(* PLC project HIBACIP, Skikda University HIBACIP CODESYS 3.5.16.50 *)
(* stored: creationDateTime 2026-06-10T00:00:00, modificationDateTime 2026-06-10T00:00:00 *)

FUNCTION_BLOCK FB_SensorDiag
  VAR_INPUT
    w_RawAI : WORD;
    r_EU_Lo : REAL;
    r_EU_Hi : REAL;
    r_Filter_Alpha : REAL := 0.15;
    r_WB_Threshold : REAL := 1000.0;
  END_VAR
  VAR_OUTPUT
    r_ScaledPV : REAL;
    r_FilteredPV : REAL;
    b_WireFault : BOOL;
    b_BadQuality : BOOL;
  END_VAR
  VAR
    r_Raw : REAL;
    r_PrevFilt : REAL;
  END_VAR

            r_Raw := WORD_TO_REAL(w_RawAI);
IF r_Raw < r_WB_Threshold THEN
    b_WireFault  := TRUE;
    b_BadQuality := TRUE;
    r_ScaledPV   := -999.0;
    r_FilteredPV := -999.0;
    RETURN;
END_IF
b_WireFault := FALSE;
r_ScaledPV  := (r_Raw / 32767.0) * (r_EU_Hi - r_EU_Lo) + r_EU_Lo;
IF r_ScaledPV > r_EU_Hi THEN r_ScaledPV := r_EU_Hi; END_IF
IF r_ScaledPV < r_EU_Lo THEN r_ScaledPV := r_EU_Lo; END_IF
r_FilteredPV := r_Filter_Alpha * r_ScaledPV
    + (1.0 - r_Filter_Alpha) * r_PrevFilt;
r_PrevFilt   := r_FilteredPV;
b_BadQuality := b_WireFault;
          
END_FUNCTION_BLOCK

FUNCTION_BLOCK FB_ValveControl
  VAR_INPUT
    b_Open_Cmd : BOOL;
    b_EStop : BOOL;
    b_FailOpen : BOOL := FALSE;
  END_VAR
  VAR_OUTPUT
    q_ValveCoil : BOOL;
  END_VAR

            IF b_EStop THEN
    q_ValveCoil := b_FailOpen;
    RETURN;
END_IF
q_ValveCoil := b_Open_Cmd;
          
END_FUNCTION_BLOCK

FUNCTION_BLOCK FB_PumpControl
  VAR_INPUT
    b_Start_Cmd : BOOL;
    b_Overload_OK : BOOL;
    b_EStop : BOOL;
  END_VAR
  VAR_OUTPUT
    q_PumpCoil : BOOL;
    b_Running : BOOL;
    b_Fault : BOOL;
  END_VAR

            IF b_EStop OR NOT b_Overload_OK THEN
    q_PumpCoil := FALSE;
    b_Running  := FALSE;
    b_Fault    := NOT b_Overload_OK;
    RETURN;
END_IF
q_PumpCoil := b_Start_Cmd;
b_Running  := q_PumpCoil;
b_Fault    := FALSE;
          
END_FUNCTION_BLOCK

FUNCTION_BLOCK FB_AlarmManager
  VAR_INPUT
    b_AlarmIn : BOOL;
    b_Ack_Cmd : BOOL;
    n_Priority : INT := 3;
  END_VAR
  VAR_OUTPUT
    b_Active : BOOL;
    b_Unacknowledged : BOOL;
  END_VAR
  VAR
    b_PrevAlarm : BOOL;
  END_VAR

            IF b_AlarmIn AND NOT b_PrevAlarm THEN
    b_Active         := TRUE;
    b_Unacknowledged := TRUE;
END_IF
b_PrevAlarm := b_AlarmIn;
IF NOT b_AlarmIn THEN b_Active := FALSE; END_IF
IF b_Ack_Cmd THEN b_Unacknowledged := FALSE; END_IF
          
END_FUNCTION_BLOCK

FUNCTION_BLOCK FB_RecipeManager
  VAR_INPUT
    n_SelectRecipe : INT := 1;
    b_Load_Cmd : BOOL;
  END_VAR
  VAR_OUTPUT
    r_Alk_Temp : REAL;
    r_Acid_Temp : REAL;
    r_Dur_AlkWash : REAL;
    r_Dur_AcidWash : REAL;
    r_Cond_Gate : REAL;
    s_RecipeName : STRING;
    n_ActiveRecipe : INT;
  END_VAR

            IF b_Load_Cmd AND n_SelectRecipe >= 1 AND n_SelectRecipe <= 4 THEN
    CASE n_SelectRecipe OF
    1: r_Alk_Temp:=30.0; r_Acid_Temp:=40.0;
       r_Dur_AlkWash:=2520.0; r_Dur_AcidWash:=1620.0;
       r_Cond_Gate:=0.5; s_RecipeName:='STD-DESCALE';
    2: r_Alk_Temp:=35.0; r_Acid_Temp:=45.0;
       r_Dur_AlkWash:=3000.0; r_Dur_AcidWash:=1800.0;
       r_Cond_Gate:=0.5; s_RecipeName:='HEAVY-SCALE';
    3: r_Alk_Temp:=25.0; r_Acid_Temp:=35.0;
       r_Dur_AlkWash:=1800.0; r_Dur_AcidWash:=1200.0;
       r_Cond_Gate:=0.5; s_RecipeName:='LIGHT-MAINT';
    4: r_Alk_Temp:=30.0; r_Acid_Temp:=40.0;
       r_Dur_AlkWash:=2700.0; r_Dur_AcidWash:=1800.0;
       r_Cond_Gate:=0.3; s_RecipeName:='PHARMA-GRADE';
    END_CASE;
    n_ActiveRecipe := n_SelectRecipe;
END_IF
          
END_FUNCTION_BLOCK

FUNCTION_BLOCK FB_PID_Industrial
  VAR_INPUT
    r_SP : REAL;
    r_PV : REAL;
    b_Auto : BOOL;
    r_Manual_Out : REAL;
    r_Kp : REAL := 3.5;
    r_Ti : REAL := 12.5;
    r_Td : REAL := 6.25;
    r_Tf : REAL := 0.5;
    r_Dt : REAL := 0.02;
    r_OutMin : REAL := 0.0;
    r_OutMax : REAL := 100.0;
  END_VAR
  VAR_OUTPUT
    r_Output : REAL;
    r_Error : REAL;
  END_VAR
  VAR
    r_Integral : REAL;
    r_D_Filt : REAL;
    r_PrevPV : REAL;
    r_Raw_Out : REAL;
    r_BackCalc : REAL;
    r_Ki : REAL;
    r_Kb : REAL;
  END_VAR

            IF NOT b_Auto THEN
    r_Output   := MAX(r_OutMin, MIN(r_OutMax, r_Manual_Out));
    r_Integral := r_Output;
    r_PrevPV   := r_PV;
    r_D_Filt   := 0.0;
    RETURN;
END_IF
r_Ki := (1.0 / r_Ti) * r_Dt;
r_Kb := r_Dt / r_Ti;
r_Error   := r_SP - r_PV;
r_Integral := r_Integral + r_Kp * r_Ki * r_Error + r_BackCalc;
r_D_Filt   := (r_Td * (r_PrevPV - r_PV) / r_Dt + r_D_Filt * r_Tf) / (r_Tf + r_Dt);
r_Raw_Out  := r_Kp * r_Error + r_Integral + r_Kp * r_D_Filt;
IF r_Raw_Out > r_OutMax THEN
    r_Output := r_OutMax;
ELSIF r_Raw_Out < r_OutMin THEN
    r_Output := r_OutMin;
ELSE
    r_Output := r_Raw_Out;
END_IF
r_BackCalc := r_Kb * (r_Output - r_Raw_Out);
r_PrevPV   := r_PV;
          
END_FUNCTION_BLOCK

FUNCTION_BLOCK FB_SafetyManager
  VAR_INPUT
    r_Temp_PV : REAL;
    r_Pressure_PV : REAL;
    r_Flow_PV : REAL;
    b_EStop_NC : BOOL;
    b_Pump_Cmd : BOOL;
    b_Pump_RunFB : BOOL;
    b_Pump_OL_OK : BOOL;
    b_AI_Temp_Fault : BOOL;
    b_AI_Pres_Fault : BOOL;
    b_SafetyReset : BOOL;
    r_Temp_TripSP : REAL := 60.0;
    r_Pres_TripSP : REAL := 6.0;
    t_PumpTimeout : TIME := T#3S;
  END_VAR
  VAR_OUTPUT
    b_EStop_Active : BOOL;
    b_Alarm_HighTemp : BOOL;
    b_Alarm_HighPres : BOOL;
    b_Alarm_LowFlow : BOOL;
    b_Alarm_PumpFault : BOOL;
    b_Alarm_AI_Fault : BOOL;
    q_SafeState_Drain : BOOL;
    n_Active : INT;
  END_VAR
  VAR
    ton_Pump : TON;
    n_Count : INT;
  END_VAR

            n_Count := 0;
IF r_Temp_PV >= r_Temp_TripSP OR b_AI_Temp_Fault THEN
    b_Alarm_HighTemp := TRUE;
    n_Count := n_Count + 1;
END_IF
IF r_Pressure_PV >= r_Pres_TripSP OR b_AI_Pres_Fault THEN
    b_Alarm_HighPres := TRUE;
    n_Count := n_Count + 1;
END_IF
ton_Pump(IN := b_Pump_Cmd AND NOT b_Pump_RunFB, PT := t_PumpTimeout);
IF ton_Pump.Q THEN
    b_Alarm_PumpFault := TRUE;
    n_Count := n_Count + 1;
END_IF
IF NOT b_EStop_NC THEN n_Count := n_Count + 1; END_IF
IF NOT b_Pump_OL_OK THEN n_Count := n_Count + 1; END_IF
b_Alarm_AI_Fault := b_AI_Temp_Fault OR b_AI_Pres_Fault;
n_Active := n_Count;
IF n_Count > 0 THEN
    b_EStop_Active    := TRUE;
    q_SafeState_Drain := TRUE;
END_IF
IF b_SafetyReset AND NOT b_Alarm_HighTemp AND NOT b_Alarm_HighPres
   AND NOT b_Alarm_PumpFault AND b_EStop_NC AND b_Pump_OL_OK THEN
    b_EStop_Active    := FALSE;
    b_Alarm_HighTemp  := FALSE;
    b_Alarm_HighPres  := FALSE;
    b_Alarm_PumpFault := FALSE;
    b_Alarm_LowFlow   := FALSE;
    q_SafeState_Drain := FALSE;
    n_Active          := 0;
END_IF
          
END_FUNCTION_BLOCK

FUNCTION_BLOCK FB_CIP
  VAR_INPUT
    cmd_Start : BOOL;
    cmd_Stop : BOOL;
    cmd_Hold : BOOL;
    cmd_Restart : BOOL;
    cmd_Abort : BOOL;
    cmd_Reset : BOOL;
    b_Permissive_OK : BOOL;
    r_Temp_PV : REAL;
    r_Cond_PV : REAL;
    r_Flow_PV : REAL;
    r_Alk_Temp_SP : REAL;
    r_Acid_Temp_SP : REAL;
    r_Cond_Baseline : REAL;
    r_Dur_InitRinse : REAL;
    r_Dur_AlkWash : REAL;
    r_Dur_InterRinse : REAL;
    r_Dur_AcidWash : REAL;
    r_Dur_FinalRinse : REAL;
  END_VAR
  VAR_OUTPUT
    q_Pump : BOOL;
    q_NaOH : BOOL;
    q_AcAc : BOOL;
    q_Rinse : BOOL;
    q_Drain : BOOL;
    q_Steam_Enable : BOOL;
    r_Temp_SP_Active : REAL;
    n_State : INT;
    n_Phase : INT;
    r_Progress : REAL;
    b_Complete : BOOL;
    b_Running : BOOL;
    b_Hold_Active : BOOL;
    b_Abort_Active : BOOL;
    s_State_Text : STRING;
    b_Alarm_Rinse_Fail : BOOL;
    r_NaOH_Vol : REAL;
    r_AcAc_Vol : REAL;
  END_VAR
  VAR
    ton_Phase : TON;
    ton_Hold : TON;
    ton_Abort : TON;
    b_TimerEN : BOOL;
    t_Target : TIME := T#3M;
    n_HoldRes : INT;
    r_Elapsed : REAL;
    r_TargetS : REAL;
  END_VAR

            IF cmd_Abort AND n_State <> 20 AND n_State <> 21 THEN
    n_State:=20; s_State_Text:='ABORTING'; b_Abort_Active:=TRUE;
    q_NaOH:=FALSE; q_AcAc:=FALSE; q_Steam_Enable:=FALSE;
    q_Drain:=TRUE; b_TimerEN:=FALSE; r_Temp_SP_Active:=0.0; RETURN;
END_IF
ton_Abort(IN:=n_State=20,PT:=T#30S);
IF ton_Abort.Q AND n_State=20 THEN
    n_State:=21; q_Drain:=FALSE; s_State_Text:='ABORTED';
END_IF
IF n_State=1 AND (NOT b_Permissive_OK OR cmd_Hold) THEN
    n_HoldRes:=n_Phase; n_State:=10; s_State_Text:='HOLDING';
    b_Hold_Active:=TRUE; b_TimerEN:=FALSE;
    q_NaOH:=FALSE; q_AcAc:=FALSE; q_Steam_Enable:=FALSE;
    q_Rinse:=TRUE; q_Pump:=TRUE;
END_IF
CASE n_State OF
0:
    q_Pump:=FALSE; q_NaOH:=FALSE; q_AcAc:=FALSE; q_Rinse:=FALSE;
    q_Drain:=FALSE; q_Steam_Enable:=FALSE; b_Complete:=FALSE;
    b_Running:=FALSE; b_Hold_Active:=FALSE; b_Abort_Active:=FALSE;
    r_Progress:=0.0; n_Phase:=0; r_Temp_SP_Active:=0.0;
    b_TimerEN:=FALSE; s_State_Text:='IDLE';
    IF cmd_Start AND b_Permissive_OK THEN
        n_State:=1; n_Phase:=1; s_State_Text:='RUNNING'; b_Running:=TRUE;
    END_IF
1:
    s_State_Text:='RUNNING'; b_Running:=TRUE;
    IF cmd_Stop THEN
        n_State:=30; b_TimerEN:=FALSE; s_State_Text:='STOPPING'; RETURN;
    END_IF
    ton_Phase(IN:=b_TimerEN,PT:=t_Target);
    r_Elapsed:=DINT_TO_REAL(TIME_TO_DINT(ton_Phase.ET))/1000.0;
    r_TargetS:=DINT_TO_REAL(TIME_TO_DINT(t_Target))/1000.0;
    IF r_TargetS > 0.0 THEN r_Progress:=MIN(100.0,r_Elapsed/r_TargetS*100.0); END_IF
    CASE n_Phase OF
    1:
        q_Rinse:=TRUE; q_Pump:=TRUE; q_Drain:=TRUE;
        q_NaOH:=FALSE; q_AcAc:=FALSE; q_Steam_Enable:=FALSE; r_Temp_SP_Active:=0.0;
        t_Target:=DINT_TO_TIME(REAL_TO_DINT(r_Dur_InitRinse*1000.0));
        IF NOT b_TimerEN THEN b_TimerEN:=TRUE; END_IF
        IF ton_Phase.Q THEN
            b_TimerEN:=FALSE; q_Drain:=FALSE; n_Phase:=2;
            ton_Phase(IN:=FALSE,PT:=t_Target);
        END_IF
    2:
        q_NaOH:=TRUE; q_Pump:=TRUE; q_Steam_Enable:=TRUE;
        q_Rinse:=FALSE; q_AcAc:=FALSE; q_Drain:=FALSE;
        r_Temp_SP_Active:=r_Alk_Temp_SP;
        t_Target:=DINT_TO_TIME(REAL_TO_DINT(r_Dur_AlkWash*1000.0));
        IF NOT b_TimerEN THEN b_TimerEN:=TRUE; END_IF
        IF ton_Phase.Q THEN
            b_TimerEN:=FALSE; q_Steam_Enable:=FALSE; r_Temp_SP_Active:=0.0; n_Phase:=3;
            ton_Phase(IN:=FALSE,PT:=t_Target);
        END_IF
    3:
        q_Rinse:=TRUE; q_Pump:=TRUE; q_Drain:=TRUE;
        q_NaOH:=FALSE; q_AcAc:=FALSE; q_Steam_Enable:=FALSE; r_Temp_SP_Active:=0.0;
        t_Target:=DINT_TO_TIME(REAL_TO_DINT(r_Dur_InterRinse*1000.0));
        IF NOT b_TimerEN THEN b_TimerEN:=TRUE; END_IF
        IF ton_Phase.Q THEN
            b_TimerEN:=FALSE; q_Drain:=FALSE; n_Phase:=4;
            ton_Phase(IN:=FALSE,PT:=t_Target);
        END_IF
    4:
        q_AcAc:=TRUE; q_Pump:=TRUE; q_Steam_Enable:=TRUE;
        q_Rinse:=FALSE; q_NaOH:=FALSE; q_Drain:=FALSE;
        r_Temp_SP_Active:=r_Acid_Temp_SP;
        t_Target:=DINT_TO_TIME(REAL_TO_DINT(r_Dur_AcidWash*1000.0));
        IF NOT b_TimerEN THEN b_TimerEN:=TRUE; END_IF
        IF ton_Phase.Q THEN
            b_TimerEN:=FALSE; q_Steam_Enable:=FALSE; r_Temp_SP_Active:=0.0; n_Phase:=5;
            ton_Phase(IN:=FALSE,PT:=t_Target);
        END_IF
    5:
        q_Rinse:=TRUE; q_Pump:=TRUE; q_Drain:=TRUE;
        q_AcAc:=FALSE; q_Steam_Enable:=FALSE; r_Temp_SP_Active:=0.0;
        t_Target:=DINT_TO_TIME(REAL_TO_DINT(r_Dur_FinalRinse*1000.0));
        IF NOT b_TimerEN THEN b_TimerEN:=TRUE; END_IF
        IF ton_Phase.Q THEN
            b_TimerEN:=FALSE; ton_Phase(IN:=FALSE,PT:=t_Target);
            IF r_Cond_PV <= r_Cond_Baseline THEN
                n_State:=5; n_Phase:=0; b_Complete:=TRUE; b_Running:=FALSE;
                r_Progress:=100.0; s_State_Text:='COMPLETE';
            ELSE
                b_Alarm_Rinse_Fail:=TRUE; n_State:=20;
                b_Abort_Active:=TRUE; s_State_Text:='ABORTING';
            END_IF
        END_IF
    END_CASE
5:
    s_State_Text:='COMPLETE'; b_Complete:=TRUE; b_Running:=FALSE;
    q_Pump:=FALSE; q_Rinse:=FALSE; q_Drain:=FALSE;
    IF cmd_Reset THEN
        n_State:=0; b_Complete:=FALSE; r_NaOH_Vol:=0.0; r_AcAc_Vol:=0.0;
        b_Alarm_Rinse_Fail:=FALSE; s_State_Text:='IDLE';
    END_IF
10:
    s_State_Text:='HOLDING'; q_Pump:=TRUE; q_Rinse:=TRUE;
    q_NaOH:=FALSE; q_AcAc:=FALSE; q_Steam_Enable:=FALSE;
    ton_Hold(IN:=TRUE,PT:=T#5S);
    IF ton_Hold.Q THEN n_State:=11; s_State_Text:='HELD'; END_IF
11:
    s_State_Text:='HELD'; q_Pump:=TRUE; q_Rinse:=TRUE;
    IF cmd_Restart AND b_Permissive_OK THEN
        n_State:=12; s_State_Text:='RESTARTING';
        b_Hold_Active:=FALSE; ton_Hold(IN:=FALSE,PT:=T#5S);
    END_IF
12:
    s_State_Text:='RESTARTING'; ton_Hold(IN:=TRUE,PT:=T#5S);
    IF ton_Hold.Q AND b_Permissive_OK THEN
        n_Phase:=n_HoldRes; n_State:=1; s_State_Text:='RUNNING'; b_TimerEN:=FALSE;
    END_IF
20:
    s_State_Text:='ABORTING'; q_NaOH:=FALSE; q_AcAc:=FALSE;
    q_Steam_Enable:=FALSE; q_Pump:=TRUE; q_Rinse:=TRUE; q_Drain:=TRUE;
21:
    s_State_Text:='ABORTED'; q_Pump:=FALSE; q_Rinse:=FALSE; q_Drain:=FALSE;
    IF cmd_Reset THEN
        b_Abort_Active:=FALSE; b_Alarm_Rinse_Fail:=FALSE;
        n_State:=0; s_State_Text:='IDLE';
    END_IF
30:
    s_State_Text:='STOPPING'; q_NaOH:=FALSE; q_AcAc:=FALSE;
    q_Steam_Enable:=FALSE; q_Pump:=TRUE; q_Rinse:=TRUE;
    ton_Hold(IN:=TRUE,PT:=T#30S);
    IF ton_Hold.Q THEN
        q_Pump:=FALSE; q_Rinse:=FALSE; n_State:=31; s_State_Text:='STOPPED';
    END_IF
31:
    s_State_Text:='STOPPED'; b_Running:=FALSE;
    IF cmd_Reset THEN n_State:=0; s_State_Text:='IDLE'; END_IF
ELSE
    GVL_Alarms.b_EStop_Active:=TRUE;
END_CASE
          
END_FUNCTION_BLOCK

PROGRAM PLC_PRG
  VAR
    fbSensTemp : FB_SensorDiag;
    fbSensPres : FB_SensorDiag;
    fbSensFlow : FB_SensorDiag;
    fbSensCond : FB_SensorDiag;
    fbSafety : FB_SafetyManager;
    fbPID : FB_PID_Industrial;
    fbCIP : FB_CIP;
    b_Permissive_OK : BOOL;
    b_PID_Auto : BOOL;
  END_VAR

            fbSensTemp(w_RawAI:=GVL_IO.w_Temp_RawAI,r_EU_Lo:=0.0,r_EU_Hi:=100.0);
GVL_IO.r_Temp_PV := fbSensTemp.r_FilteredPV;
fbSensPres(w_RawAI:=GVL_IO.w_Pres_RawAI,r_EU_Lo:=0.0,r_EU_Hi:=10.0);
GVL_IO.r_Pres_PV := fbSensPres.r_FilteredPV;
fbSensFlow(w_RawAI:=GVL_IO.w_Flow_RawAI,r_EU_Lo:=0.0,r_EU_Hi:=100.0);
GVL_IO.r_Flow_PV := fbSensFlow.r_FilteredPV;
fbSensCond(w_RawAI:=GVL_IO.w_Cond_RawAI,r_EU_Lo:=0.0,r_EU_Hi:=20.0);
GVL_IO.r_Cond_PV := fbSensCond.r_FilteredPV;
GVL_IO.i_CircPump_RunFB := GVL_IO.q_CircPump;
fbSafety(
    r_Temp_PV:=GVL_IO.r_Temp_PV, r_Pressure_PV:=GVL_IO.r_Pres_PV,
    r_Flow_PV:=GVL_IO.r_Flow_PV, b_EStop_NC:=GVL_IO.i_EStop_NC,
    b_Pump_Cmd:=GVL_IO.q_CircPump, b_Pump_RunFB:=GVL_IO.i_CircPump_RunFB,
    b_Pump_OL_OK:=GVL_IO.i_CircPump_OL,
    b_AI_Temp_Fault:=fbSensTemp.b_WireFault,
    b_AI_Pres_Fault:=fbSensPres.b_WireFault,
    b_SafetyReset:=GVL_IO.i_SafetyReset);
IF fbSafety.b_EStop_Active THEN
    GVL_IO.q_CircPump:=FALSE; GVL_IO.q_NaOH_Valve:=FALSE;
    GVL_IO.q_AcAc_Valve:=FALSE; GVL_IO.q_Rinse_Valve:=FALSE;
    GVL_IO.q_Steam_Enable:=FALSE; GVL_IO.q_Drain_Valve:=TRUE;
    GVL_IO.r_SteamValve_Pct:=0.0; GVL_IO.q_Alarm_Light_R:=TRUE;
    GVL_Alarms.b_EStop_Active:=TRUE;
    GVL_Alarms.s_State_Name:='E-STOP'; RETURN;
END_IF
GVL_Alarms.b_EStop_Active:=FALSE;
GVL_IO.q_Alarm_Light_R:=FALSE;
b_Permissive_OK :=
    GVL_IO.i_FlowSwitch_Min AND GVL_IO.i_EStop_NC AND GVL_IO.i_CircPump_OL
    AND NOT fbSensTemp.b_WireFault AND (GVL_IO.r_Flow_PV > 0.0)
    AND (GVL_IO.r_Temp_PV < GVL_Setpoints.r_Temp_HighTrip - 10.0);
IF fbCIP.n_State = 1 THEN GVL_IO.i_Start_Command := FALSE; END_IF
IF fbCIP.n_State = 31 THEN GVL_HMI.b_Stop_Cmd := FALSE; END_IF
IF fbCIP.n_State = 0 THEN GVL_HMI.b_Reset_Cmd := FALSE; END_IF
fbCIP(
    cmd_Start:=GVL_IO.i_Start_Command, cmd_Stop:=GVL_HMI.b_Stop_Cmd,
    cmd_Hold:=GVL_HMI.b_Hold_Cmd, cmd_Restart:=GVL_HMI.b_Restart_Cmd,
    cmd_Abort:=GVL_HMI.b_Abort_Cmd, cmd_Reset:=GVL_HMI.b_Reset_Cmd,
    b_Permissive_OK:=b_Permissive_OK,
    r_Temp_PV:=GVL_IO.r_Temp_PV, r_Cond_PV:=GVL_IO.r_Cond_PV,
    r_Flow_PV:=GVL_IO.r_Flow_PV,
    r_Alk_Temp_SP:=GVL_Setpoints.r_Alk_Temp_SP,
    r_Acid_Temp_SP:=GVL_Setpoints.r_Acid_Temp_SP,
    r_Cond_Baseline:=GVL_Setpoints.r_Cond_Baseline,
    r_Dur_InitRinse:=GVL_Setpoints.r_Dur_InitRinse,
    r_Dur_AlkWash:=GVL_Setpoints.r_Dur_AlkWash,
    r_Dur_InterRinse:=GVL_Setpoints.r_Dur_InterRinse,
    r_Dur_AcidWash:=GVL_Setpoints.r_Dur_AcidWash,
    r_Dur_FinalRinse:=GVL_Setpoints.r_Dur_FinalRinse);
GVL_IO.q_CircPump:=fbCIP.q_Pump; GVL_IO.q_NaOH_Valve:=fbCIP.q_NaOH;
GVL_IO.q_AcAc_Valve:=fbCIP.q_AcAc; GVL_IO.q_Rinse_Valve:=fbCIP.q_Rinse;
GVL_IO.q_Drain_Valve:=fbCIP.q_Drain; GVL_IO.q_Steam_Enable:=fbCIP.q_Steam_Enable;
GVL_Alarms.n_CIP_State:=fbCIP.n_State; GVL_Alarms.n_CIP_Phase:=fbCIP.n_Phase;
GVL_Alarms.r_Phase_Progress:=fbCIP.r_Progress;
GVL_Alarms.s_State_Name:=fbCIP.s_State_Text;
GVL_Alarms.b_CIP_Complete:=fbCIP.b_Complete;
GVL_Alarms.b_Hold_Active:=fbCIP.b_Hold_Active;
b_PID_Auto := GVL_IO.q_Steam_Enable;
fbPID(r_SP:=fbCIP.r_Temp_SP_Active, r_PV:=GVL_IO.r_Temp_PV,
    b_Auto:=b_PID_Auto, r_Manual_Out:=GVL_HMI.r_PID_ManualOut,
    r_Kp:=GVL_Setpoints.r_PID_Kp, r_Ti:=GVL_Setpoints.r_PID_Ti,
    r_Td:=GVL_Setpoints.r_PID_Td, r_Tf:=GVL_Setpoints.r_PID_Tf,
    r_Dt:=GVL_Setpoints.r_PID_Dt);
GVL_IO.r_SteamValve_Pct:=fbPID.r_Output;
GVL_IO.w_SteamValve_AO:=REAL_TO_WORD(GVL_IO.r_SteamValve_Pct/100.0*32767.0);
GVL_IO.q_Status_Light_G:=fbCIP.b_Running;
          
END_PROGRAM

CONFIGURATION HIBACIP
  RESOURCE Resource ON PLC
    VAR_GLOBAL  (* GVL_IO *)
      w_Temp_RawAI : WORD := 7209;
      w_Pres_RawAI : WORD := 6554;
      w_Flow_RawAI : WORD := 8192;
      w_Cond_RawAI : WORD := 1311;
      r_Temp_PV : REAL;
      r_Pres_PV : REAL;
      r_Flow_PV : REAL;
      r_Cond_PV : REAL;
      i_Start_Command : BOOL := FALSE;
      i_EStop_NC : BOOL := TRUE;
      i_CircPump_RunFB : BOOL := FALSE;
      i_CircPump_OL : BOOL := TRUE;
      i_FlowSwitch_Min : BOOL := TRUE;
      i_SafetyReset : BOOL := FALSE;
      q_CircPump : BOOL := FALSE;
      q_NaOH_Valve : BOOL := FALSE;
      q_AcAc_Valve : BOOL := FALSE;
      q_Rinse_Valve : BOOL := FALSE;
      q_Drain_Valve : BOOL := FALSE;
      q_Steam_Enable : BOOL := FALSE;
      q_Alarm_Light_R : BOOL := FALSE;
      q_Status_Light_G : BOOL := FALSE;
      q_Alarm_Horn : BOOL := FALSE;
      r_SteamValve_Pct : REAL;
      w_SteamValve_AO : WORD;
    END_VAR
    VAR_GLOBAL RETAIN  (* GVL_Setpoints *)
      r_Alk_Temp_SP : REAL := 30.0;
      r_Acid_Temp_SP : REAL := 40.0;
      r_Temp_HighTrip : REAL := 60.0;
      r_Cond_Baseline : REAL := 0.5;
      r_Dur_InitRinse : REAL := 180.0;
      r_Dur_AlkWash : REAL := 2520.0;
      r_Dur_InterRinse : REAL := 180.0;
      r_Dur_AcidWash : REAL := 1620.0;
      r_Dur_FinalRinse : REAL := 300.0;
      r_PID_Kp : REAL := 3.5;
      r_PID_Ti : REAL := 12.5;
      r_PID_Td : REAL := 6.25;
      r_PID_Tf : REAL := 0.5;
      r_PID_Dt : REAL := 0.02;
    END_VAR
    VAR_GLOBAL  (* GVL_Alarms *)
      b_EStop_Active : BOOL := FALSE;
      b_Alarm_HighTemp : BOOL := FALSE;
      b_Alarm_HighPres : BOOL := FALSE;
      b_Alarm_PumpFault : BOOL := FALSE;
      b_Alarm_RinseFail : BOOL := FALSE;
      n_CIP_State : INT;
      n_CIP_Phase : INT;
      r_Phase_Progress : REAL;
      b_CIP_Complete : BOOL := FALSE;
      b_Hold_Active : BOOL := FALSE;
      s_State_Name : STRING;
    END_VAR
    VAR_GLOBAL  (* GVL_HMI *)
      b_Stop_Cmd : BOOL := FALSE;
      b_Hold_Cmd : BOOL := FALSE;
      b_Restart_Cmd : BOOL := FALSE;
      b_Abort_Cmd : BOOL := FALSE;
      b_Reset_Cmd : BOOL := FALSE;
      b_HornSilence : BOOL := FALSE;
      r_PID_ManualOut : REAL;
    END_VAR
    TASK MainTask(INTERVAL := T#20ms, PRIORITY := 1);
    PROGRAM PLC_PRG WITH MainTask : PLC_PRG;
  END_RESOURCE
END_CONFIGURATION
